FUNCTION_BLOCK Delay_With_InitCondition (* Composite Function Block Type *)
  (* Standard: 61499-2; Description: INIT nya disambungin ke start/warm cold yaa Trus conf nya ntar dibalikin lagi ke Start_and_REQ juga *)
  (* Version 0.0, 2018-07-28, 4DIAC-IDE, 4DIAC-Consortium *)
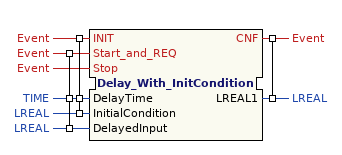
  EVENT_INPUT
    INIT WITH DelayTime, InitialCondition;
    Start_and_REQ WITH DelayTime, DelayedInput; (* Normal Execution Request *)
    Stop;
  END_EVENT
  EVENT_OUTPUT
    CNF WITH LREAL1; (* Execution Confirmation *)
  END_EVENT
  VAR_INPUT
    DelayTime : TIME;
    InitialCondition : LREAL;
    DelayedInput : LREAL;
  END_VAR
  VAR_OUTPUT
    LREAL1 : LREAL;
  END_VAR
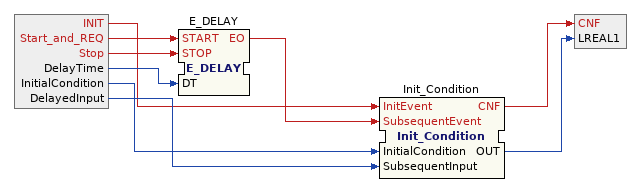
  FBS
    E_DELAY : E_DELAY;
    Init_Condition : Init_Condition;
  END_FBS
  EVENT_CONNECTIONS
    Start_and_REQ TO E_DELAY.START;
    Stop TO E_DELAY.STOP;
    INIT TO Init_Condition.InitEvent;
    E_DELAY.EO TO Init_Condition.SubsequentEvent;
    Init_Condition.CNF TO CNF;
  END_CONNECTIONS
  DATA_CONNECTIONS
    DelayTime TO E_DELAY.DT;
    Init_Condition.OUT TO LREAL1;
    DelayedInput TO Init_Condition.SubsequentInput;
    InitialCondition TO Init_Condition.InitialCondition;
  END_CONNECTIONS
END_FUNCTION_BLOCK
